(* Logix 5000 project; controller test vendor 1 type 14 code 196 rev 35.11; software revision 35.00 *)

TASK MainTask (continuous, watchdog 500 ms) : MainProgram

MODULES
   Local : vendor 1 type 14 code 196 (5069 0, rev 35.11)
END_MODULES

PROGRAM MainProgram   (* main routine MainRoutine *)
VAR
   Check_with_sensor : BOOL;
   Debarking_left_sensor : BOOL;
   Debarking_motor : BOOL;
   Debarking_rail_left : BOOL;
   Debarking_right_sensor : BOOL;
   Emergency : BOOL;
   Emergency_Stop_1 : BOOL;
   Emergency_Stop_2 : BOOL;
   Log_debarked : BOOL;
   Log_in_position : BOOL;
   Log_Unloaded : BOOL;
   Motor_speed : DINT;
   Move_to_left : BOOL;
   Move_to_right : BOOL;
   Process : DINT;
   Put_Log_in : BOOL;
   Release_log : BOOL;
   Running : BOOL;
   Start_Process : BOOL;
   VFD_Frequency : DINT;
   Visual_sensor : BOOL;
END_VAR

ROUTINE MainRoutine   (* ladder *)
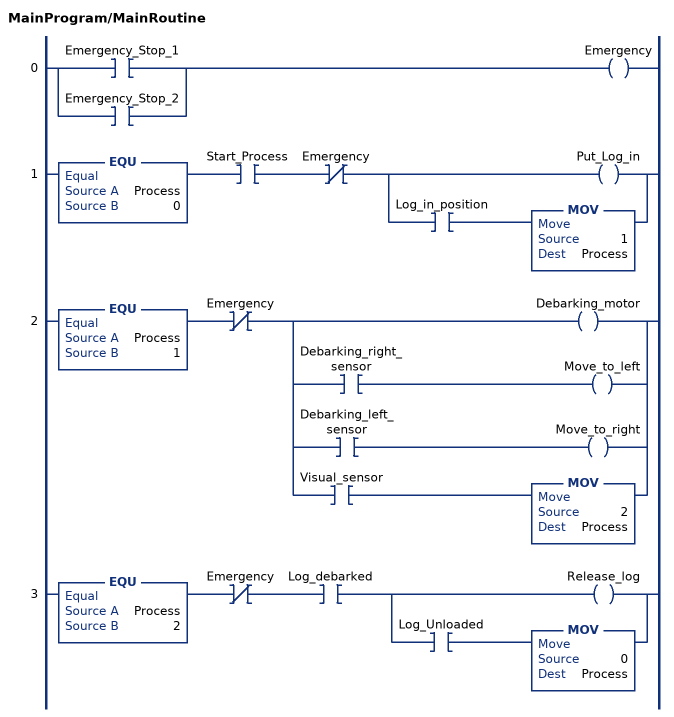
   0: [XIC(Emergency_Stop_1) ,XIC(Emergency_Stop_2) ]OTE(Emergency);
   1: EQU(Process,0)XIC(Start_Process)XIO(Emergency)[OTE(Put_Log_in) ,XIC(Log_in_position) MOV(1,Process) ];
   2: EQU(Process,1)XIO(Emergency)[OTE(Debarking_motor) ,XIC(Debarking_right_sensor) OTE(Move_to_left) ,XIC(Debarking_left_sensor) OTE(Move_to_right) ,XIC(Visual_sensor) MOV(2,Process) ];
   3: EQU(Process,2)XIO(Emergency)XIC(Log_debarked)[OTE(Release_log) ,XIC(Log_Unloaded) MOV(0,Process) ];
END_ROUTINE
END_PROGRAM
